TYPE (* Coherent snapshot of the cell state variables (contract vocabulary) *)
  (* Standard: 61499-2 *)
  (* Version 2.0, 2026-09-27, Project contributors, Filling cell reference model *)
  PACKAGE fillingcell;
  ST_CellState : STRUCT
    NeedleUp : BOOL;
    NeedleDown : BOOL;
    VialPresent : BOOL;
    FilledMl : LREAL;
    Stoppered : BOOL;
    Checked : BOOL;
    DoorClosed : BOOL;
    Valid : BOOL;
    Safe : BOOL;
  END_STRUCT;
END_TYPE
